FUNCTION_BLOCK FB_Measuring
VAR_INPUT
	VIn		:	REAL;
END_VAR
VAR_OUTPUT
	EndMeasure	:	BOOL;
	
END_VAR
VAR_IN_OUT
	VOut		:	REAL;
END_VAR
VAR
	VPrev	:	REAL	:=	10.0;
	fbTonEndMeasure	:	TON;
	En : BOOL;
END_VAR

//fbTonEndMeasure(IN := En = TRUE, PT := T#500MS);
//EndMeasure := fbTonEndMeasure.Q;
IF VIn < VPrev THEN
	VPrev := VIn;
	En := TRUE;
END_IF
IF VIn > 7.3 THEN
	Vprev := VIn;
	En := FALSE;
END_IF
IF En = TRUE THEN
	Vout:=VPrev;
END_IF

END_FUNCTION_BLOCK

(* stored: Version 1.1.0.1, ProductVersion 3.1.4024.12
   POU FB_Measuring: Id {f75dd6fc-0bf7-48b8-9633-3a5a68e2bc81}, SpecialFunc None *)
